Omron CX-Programmer project NewProject (CX-Programmer 9.75)

# PLC cj1m_cpu22: CJ1M CPU11

## Global symbols (name address type ; comment)
ActualPosition_Y _NCCPU204_ReadActualPosition_REAL
101.00 BOOL  ; Coolant Pump On
101.01 BOOL  ; X Lube Pump On
101.02 BOOL  ; Main Pump On
101.03 BOOL  ; Spindle Lube Pump On
101.04 BOOL  ; SP Main Contactor On
101.05 BOOL  ; SP Delta Contactor On
101.06 BOOL  ; SP Star Contactor On
101.07 BOOL  ; Work Light On
101.08 BOOL  ; Red Tower Light On
101.09 BOOL  ; Greeen Tower Light On
101.10 BOOL  ; Yellow Tower Light On
101.11 BOOL  ; X + Move Solenoid
101.12 BOOL  ; X - Move Solenoid
101.13 BOOL  ; X Slow Speed Solenoid
101.14 BOOL  ; X Pressure Relief Solenoid
102.00 BOOL  ; Table Magnet On
102.01 BOOL  ; Table Demagnet On
1.00 BOOL  ; Emergency PB
1.01 BOOL  ; X + PB
1.02 BOOL  ; X - PB
1.03 BOOL  ; X Stop PB
1.04 BOOL  ; Man/Auto SW
1.05 BOOL  ; Coolant Pump Overload Input
1.06 BOOL  ; X Lube Pump Overload Input
1.07 BOOL  ; Main Pump Overload Input
1.08 BOOL  ; Counterbalance Pump Overload Input
1.09 BOOL  ; Spindle Lube Pump Overload Input
1.10 BOOL  ; Spindle Chiller Overload Input
1.11 BOOL  ; Main Chiller Overload Input
1.14 BOOL  ; Alarm Y Axis Input
1.15 BOOL  ; Alarm Z Axis Input
2.00 BOOL  ; X Axis Handwheel Input
2.01 BOOL  ; Y Axis Handwheel Input
2.02 BOOL  ; Z Axis Handwheel Input
2.03 BOOL  ; X1 Speed Input
2.04 BOOL  ; X10 Speed Input
2.05 BOOL  ; X100 Speed Input
2.06 BOOL  ; X+ Work Limit SW
2.07 BOOL  ; X - Work Limit SW
2.08 BOOL  ; X + Safety Limit SW
2.09 BOOL  ; X - Safety Limit SW
2.10 BOOL  ; Z - Limit SW
2.11 BOOL  ; Z + Limit SW
2.12 BOOL  ; Z Zero Limit SW
2.13 BOOL  ; Y - Limit SW
2.14 BOOL  ; Y + Limit SW
2.15 BOOL  ; Y Zero Limit SW
3.00 BOOL  ; X Lube PR SW
3.01 BOOL  ; Spindle Lube PR SW
A540.08 BOOL  ; Y Axis Positive Limit
A540.09 BOOL  ; Y Axis Negative Limit
A541.08 BOOL  ; Z Axis Positive Limit
A541.09 BOOL  ; Z Axis Negative Limit
D10 CHANNEL  ; Travel Position
D100 CHANNEL  ; Axis Y Acceleration
D102 CHANNEL  ; Axis Y Deceleration
D108 CHANNEL  ; Axis Y Velocity
D110 CHANNEL  ; Y Actual Position
D112 CHANNEL  ; Y Jog Velocity
D20 CHANNEL  ; Travel Position Z Axis
D200 CHANNEL  ; Axis Z Acceleration
D202 CHANNEL  ; Axis Z Decceleration
D208 CHANNEL  ; Axis Z Velocity
D210 CHANNEL  ; Z Actual Position
D212 CHANNEL  ; Z Jog Velocity
W11.00 BOOL  ; Emergency Active
W11.01 BOOL  ; X + Move
W11.02 BOOL  ; X - Move
W11.03 BOOL  ; X Stop
W11.04 BOOL  ; Auto Mode
W11.05 BOOL  ; Coolant Pump Overload
W11.06 BOOL  ; X Lube Pump Overload
W11.07 BOOL  ; Main Pump Overload
W11.08 BOOL  ; Counterbalance Pump Overload
W11.09 BOOL  ; Spindle Lube Pump Overload
W11.10 BOOL  ; Spindle Chiller Overload
W11.11 BOOL  ; Main Chiller Overload
W11.14 BOOL  ; Alarm Y Axis
W11.15 BOOL  ; Alarm Z Axis
W12.00 BOOL  ; Handwheel X axis
W12.01 BOOL  ; Handwheel Y Axis
W12.02 BOOL  ; Handwheel Z Axis
W12.03 BOOL  ; Handwheel X1 Speed
W12.04 BOOL  ; Handwheel X10 Speed
W12.05 BOOL  ; Handwheel X100 Speed
W12.06 BOOL  ; X + Work Limit
W12.07 BOOL  ; X - Work Limit
W12.08 BOOL  ; X + Safety Limit
W12.09 BOOL  ; X - Safety Limit
W12.10 BOOL  ; Z - Limit
W12.11 BOOL  ; Z + Limit
W12.12 BOOL  ; Z Zero Limit
W12.13 BOOL  ; Y - Limit
W12.14 BOOL  ; Y + Limit
W12.15 BOOL  ; Y Zero Limit
W13.00 BOOL  ; X Lube Pressure Ok
W13.01 BOOL  ; Spindle Lube Pressure Ok
W21.00 BOOL  ; Coolant Pump On
W21.01 BOOL  ; X Lube Pump On
W21.02 BOOL  ; Main Pump On
W21.03 BOOL  ; Spindle Lube Pump On
W21.04 BOOL  ; Spindle Main Contactor On
W21.05 BOOL  ; Spindle Delta Contactor On
W21.06 BOOL  ; Spindle Star Contactor On
W21.07 BOOL  ; Work Light On
W21.08 BOOL  ; Red Tower Light
W21.09 BOOL  ; Green Tower Light
W21.10 BOOL  ; Yellow Tower Light
W21.11 BOOL  ; X + Move Command
W21.12 BOOL  ; X - Move Command
W21.13 BOOL  ; X Slow Speed Command
W21.14 BOOL  ; X Pressure Relief Command
W22.00 BOOL  ; Table Magnet On
W22.01 BOOL  ; Table Demagnet On
W30.00 BOOL  ; Y Axis Move Command
W30.04 BOOL  ; Y Axis Forward
W30.05 BOOL  ; Y Axis Backward
W31.04 BOOL  ; Z Jog Forward
W31.05 BOOL  ; Z Jog Backwards
W40.00 BOOL  ; X + Move Command
W40.01 BOOL  ; X - Move Command
W40.02 BOOL  ; X + Move Manual
W40.03 BOOL  ; X - Move Manual
JogBackwards_Y _NCCPU030_MoveVelocity_REAL
JogBackwards_Z _NCCPU030_MoveVelocity_REAL
JogForward_Y _NCCPU030_MoveVelocity_REAL
JogForward_Z _NCCPU030_MoveVelocity_REAL
MoveAbsolute_Z _NCCPU010_MoveAbsolute_REAL
MoveY _NCCPU010_MoveAbsolute_REAL
Position_Z _NCCPU204_ReadActualPosition_REAL

## Program NewProgram1 (cyclic task 0)

### Section Inputs

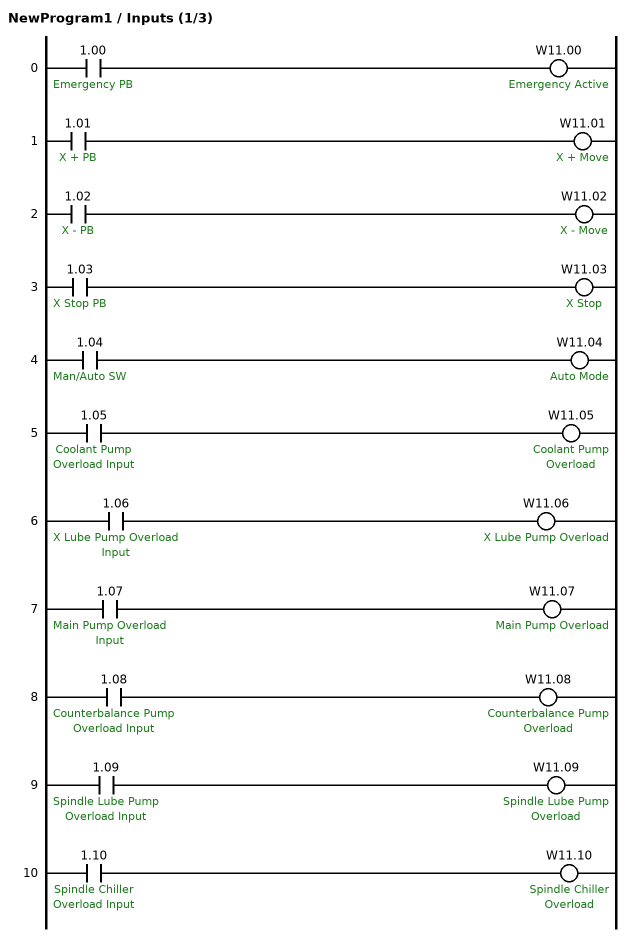
; rung 0
LD 1.00  ; Emergency PB
OUT W11.00  ; Emergency Active
; rung 1
LD 1.01  ; X + PB
OUT W11.01  ; X + Move
; rung 2
LD 1.02  ; X - PB
OUT W11.02  ; X - Move
; rung 3
LD 1.03  ; X Stop PB
OUT W11.03  ; X Stop
; rung 4
LD 1.04  ; Man/Auto SW
OUT W11.04  ; Auto Mode
; rung 5
LD 1.05  ; Coolant Pump Overload Input
OUT W11.05  ; Coolant Pump Overload
; rung 6
LD 1.06  ; X Lube Pump Overload Input
OUT W11.06  ; X Lube Pump Overload
; rung 7
LD 1.07  ; Main Pump Overload Input
OUT W11.07  ; Main Pump Overload
; rung 8
LD 1.08  ; Counterbalance Pump Overload Input
OUT W11.08  ; Counterbalance Pump Overload
; rung 9
LD 1.09  ; Spindle Lube Pump Overload Input
OUT W11.09  ; Spindle Lube Pump Overload
; rung 10
LD 1.10  ; Spindle Chiller Overload Input
OUT W11.10  ; Spindle Chiller Overload

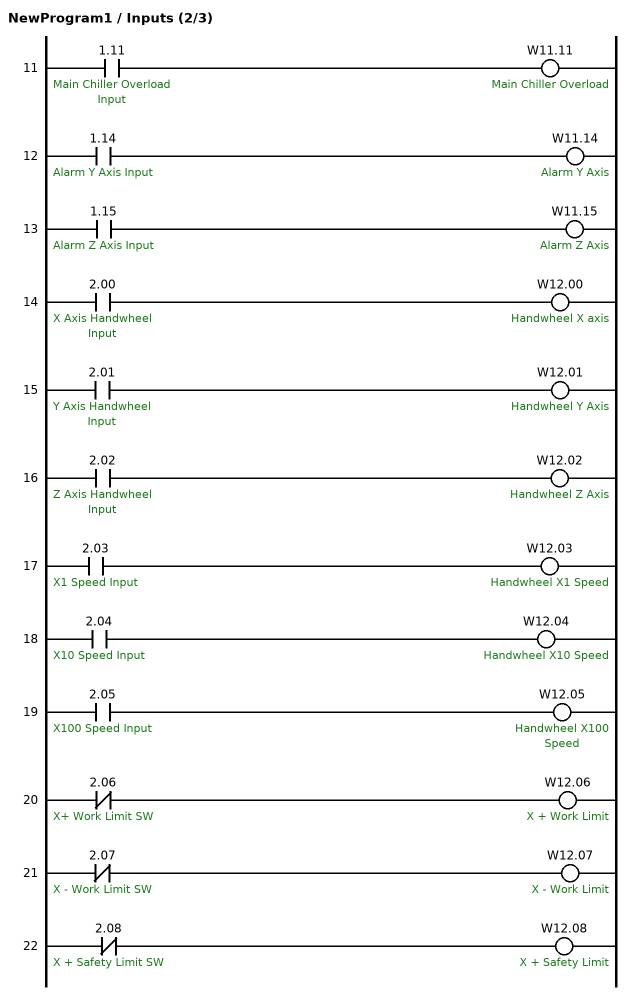
; rung 11
LD 1.11  ; Main Chiller Overload Input
OUT W11.11  ; Main Chiller Overload
; rung 12
LD 1.14  ; Alarm Y Axis Input
OUT W11.14  ; Alarm Y Axis
; rung 13
LD 1.15  ; Alarm Z Axis Input
OUT W11.15  ; Alarm Z Axis
; rung 14
LD 2.00  ; X Axis Handwheel Input
OUT W12.00  ; Handwheel X axis
; rung 15
LD 2.01  ; Y Axis Handwheel Input
OUT W12.01  ; Handwheel Y Axis
; rung 16
LD 2.02  ; Z Axis Handwheel Input
OUT W12.02  ; Handwheel Z Axis
; rung 17
LD 2.03  ; X1 Speed Input
OUT W12.03  ; Handwheel X1 Speed
; rung 18
LD 2.04  ; X10 Speed Input
OUT W12.04  ; Handwheel X10 Speed
; rung 19
LD 2.05  ; X100 Speed Input
OUT W12.05  ; Handwheel X100 Speed
; rung 20
LDNOT 2.06  ; X+ Work Limit SW
OUT W12.06  ; X + Work Limit
; rung 21
LDNOT 2.07  ; X - Work Limit SW
OUT W12.07  ; X - Work Limit
; rung 22
LDNOT 2.08  ; X + Safety Limit SW
OUT W12.08  ; X + Safety Limit

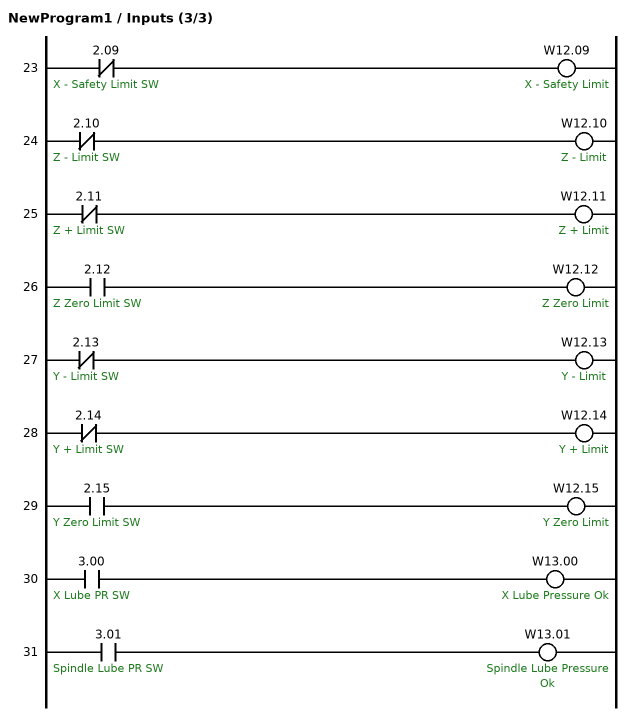
; rung 23
LDNOT 2.09  ; X - Safety Limit SW
OUT W12.09  ; X - Safety Limit
; rung 24
LDNOT 2.10  ; Z - Limit SW
OUT W12.10  ; Z - Limit
; rung 25
LDNOT 2.11  ; Z + Limit SW
OUT W12.11  ; Z + Limit
; rung 26
LD 2.12  ; Z Zero Limit SW
OUT W12.12  ; Z Zero Limit
; rung 27
LDNOT 2.13  ; Y - Limit SW
OUT W12.13  ; Y - Limit
; rung 28
LDNOT 2.14  ; Y + Limit SW
OUT W12.14  ; Y + Limit
; rung 29
LD 2.15  ; Y Zero Limit SW
OUT W12.15  ; Y Zero Limit
; rung 30
LD 3.00  ; X Lube PR SW
OUT W13.00  ; X Lube Pressure Ok
; rung 31
LD 3.01  ; Spindle Lube PR SW
OUT W13.01  ; Spindle Lube Pressure Ok

### Section Outputs

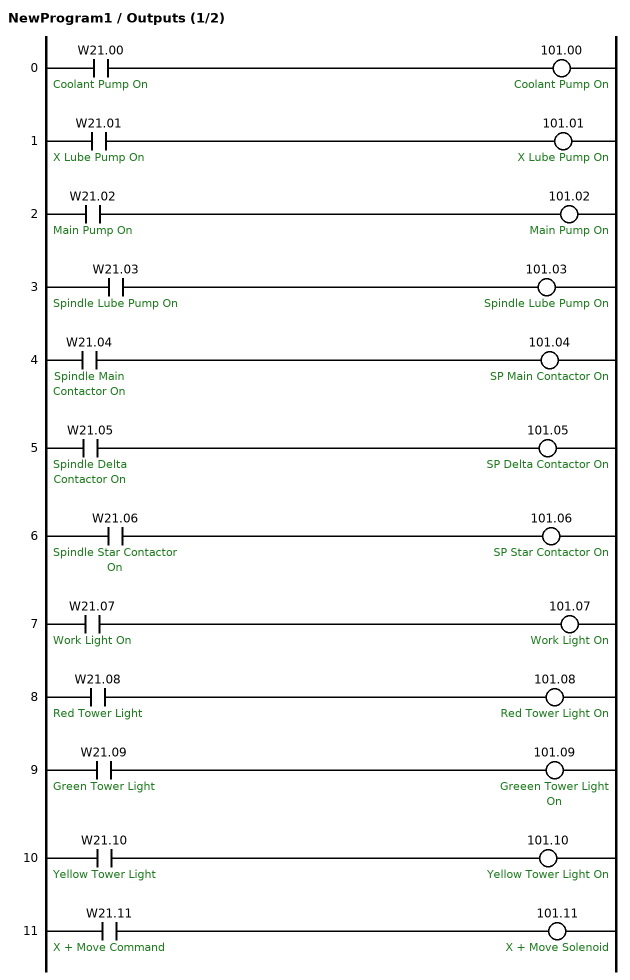
; rung 0
LD W21.00  ; Coolant Pump On
OUT 101.00  ; Coolant Pump On
; rung 1
LD W21.01  ; X Lube Pump On
OUT 101.01  ; X Lube Pump On
; rung 2
LD W21.02  ; Main Pump On
OUT 101.02  ; Main Pump On
; rung 3
LD W21.03  ; Spindle Lube Pump On
OUT 101.03  ; Spindle Lube Pump On
; rung 4
LD W21.04  ; Spindle Main Contactor On
OUT 101.04  ; SP Main Contactor On
; rung 5
LD W21.05  ; Spindle Delta Contactor On
OUT 101.05  ; SP Delta Contactor On
; rung 6
LD W21.06  ; Spindle Star Contactor On
OUT 101.06  ; SP Star Contactor On
; rung 7
LD W21.07  ; Work Light On
OUT 101.07  ; Work Light On
; rung 8
LD W21.08  ; Red Tower Light
OUT 101.08  ; Red Tower Light On
; rung 9
LD W21.09  ; Green Tower Light
OUT 101.09  ; Greeen Tower Light On
; rung 10
LD W21.10  ; Yellow Tower Light
OUT 101.10  ; Yellow Tower Light On
; rung 11
LD W21.11  ; X + Move Command
OUT 101.11  ; X + Move Solenoid

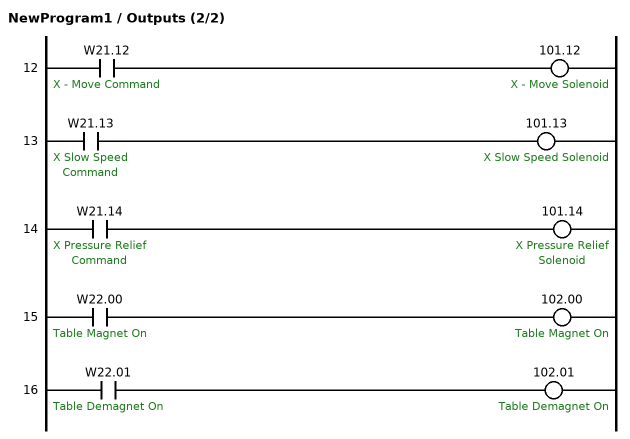
; rung 12
LD W21.12  ; X - Move Command
OUT 101.12  ; X - Move Solenoid
; rung 13
LD W21.13  ; X Slow Speed Command
OUT 101.13  ; X Slow Speed Solenoid
; rung 14
LD W21.14  ; X Pressure Relief Command
OUT 101.14  ; X Pressure Relief Solenoid
; rung 15
LD W22.00  ; Table Magnet On
OUT 102.00  ; Table Magnet On
; rung 16
LD W22.01  ; Table Demagnet On
OUT 102.01  ; Table Demagnet On

### Section Table_Movement

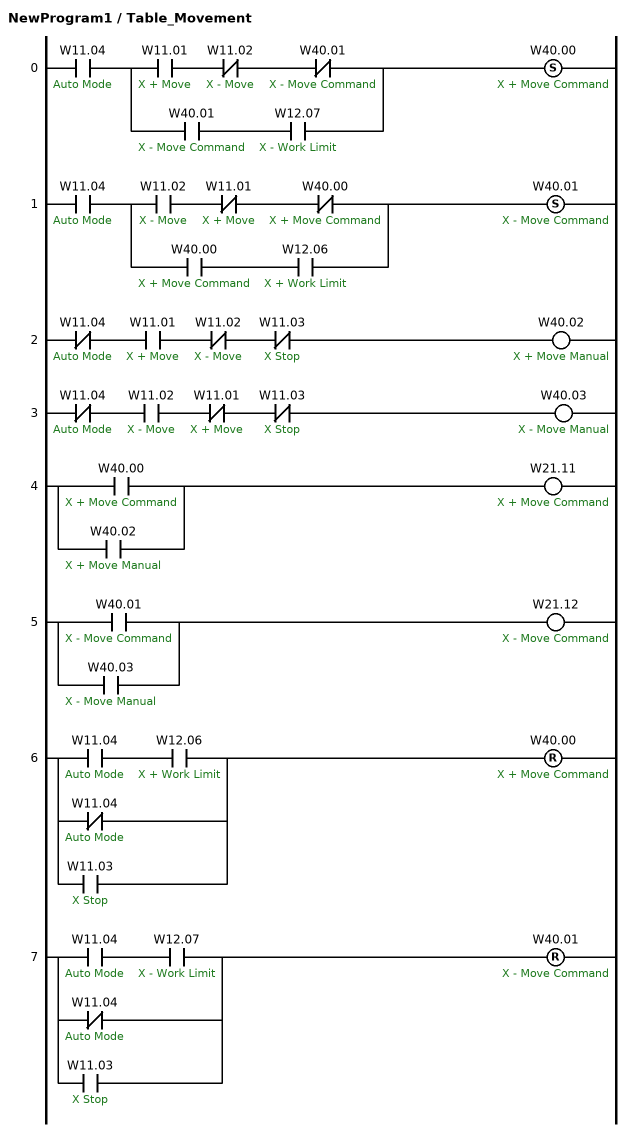
; rung 0
LD W11.04  ; Auto Mode
LD W11.01  ; X + Move
ANDNOT W11.02  ; X - Move
ANDNOT W40.01  ; X - Move Command
LD W40.01  ; X - Move Command
AND W12.07  ; X - Work Limit
ORLD
ANDLD
SET W40.00  ; X + Move Command
; rung 1
LD W11.04  ; Auto Mode
LD W11.02  ; X - Move
ANDNOT W11.01  ; X + Move
ANDNOT W40.00  ; X + Move Command
LD W40.00  ; X + Move Command
AND W12.06  ; X + Work Limit
ORLD
ANDLD
SET W40.01  ; X - Move Command
; rung 2
LDNOT W11.04  ; Auto Mode
AND W11.01  ; X + Move
ANDNOT W11.02  ; X - Move
ANDNOT W11.03  ; X Stop
OUT W40.02  ; X + Move Manual
; rung 3
LDNOT W11.04  ; Auto Mode
AND W11.02  ; X - Move
ANDNOT W11.01  ; X + Move
ANDNOT W11.03  ; X Stop
OUT W40.03  ; X - Move Manual
; rung 4
LD W40.00  ; X + Move Command
OR W40.02  ; X + Move Manual
OUT W21.11  ; X + Move Command
; rung 5
LD W40.01  ; X - Move Command
OR W40.03  ; X - Move Manual
OUT W21.12  ; X - Move Command
; rung 6
LD W11.04  ; Auto Mode
AND W12.06  ; X + Work Limit
ORNOT W11.04  ; Auto Mode
OR W11.03  ; X Stop
RSET W40.00  ; X + Move Command
; rung 7
LD W11.04  ; Auto Mode
AND W12.07  ; X - Work Limit
ORNOT W11.04  ; Auto Mode
OR W11.03  ; X Stop
RSET W40.01  ; X - Move Command

### Section Axis_Y

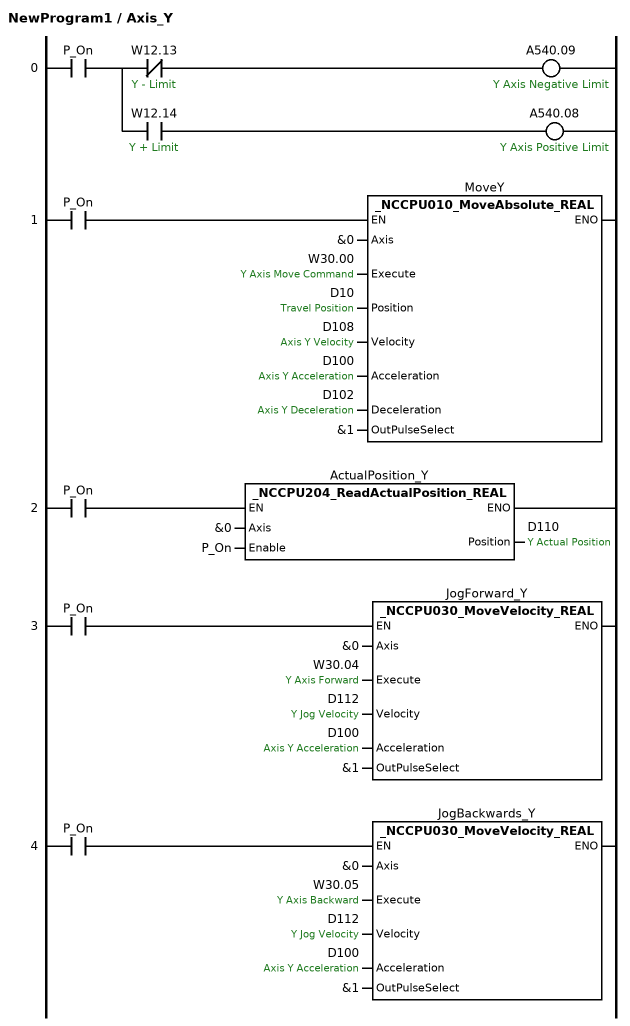
; rung 0
LD P_On
OUT TR0
ANDNOT W12.13  ; Y - Limit
OUT A540.09  ; Y Axis Negative Limit
LD TR0
AND W12.14  ; Y + Limit
OUT A540.08  ; Y Axis Positive Limit
; rung 1
LD P_On
CALL MoveY : _NCCPU010_MoveAbsolute_REAL (Axis := &0, Execute := W30.00, Position := D10, Velocity := D108, Acceleration := D100, Deceleration := D102, OutPulseSelect := &1)  ; Y Axis Move Command, Travel Position, Axis Y Velocity, Axis Y Acceleration, Axis Y Deceleration
; rung 2
LD P_On
CALL ActualPosition_Y : _NCCPU204_ReadActualPosition_REAL (Axis := &0, Enable := P_On, Position => D110)  ; Y Actual Position
; rung 3
LD P_On
CALL JogForward_Y : _NCCPU030_MoveVelocity_REAL (Axis := &0, Execute := W30.04, Velocity := D112, Acceleration := D100, OutPulseSelect := &1)  ; Y Axis Forward, Y Jog Velocity, Axis Y Acceleration
; rung 4
LD P_On
CALL JogBackwards_Y : _NCCPU030_MoveVelocity_REAL (Axis := &0, Execute := W30.05, Velocity := D112, Acceleration := D100, OutPulseSelect := &1)  ; Y Axis Backward, Y Jog Velocity, Axis Y Acceleration

### Section Axis_Z

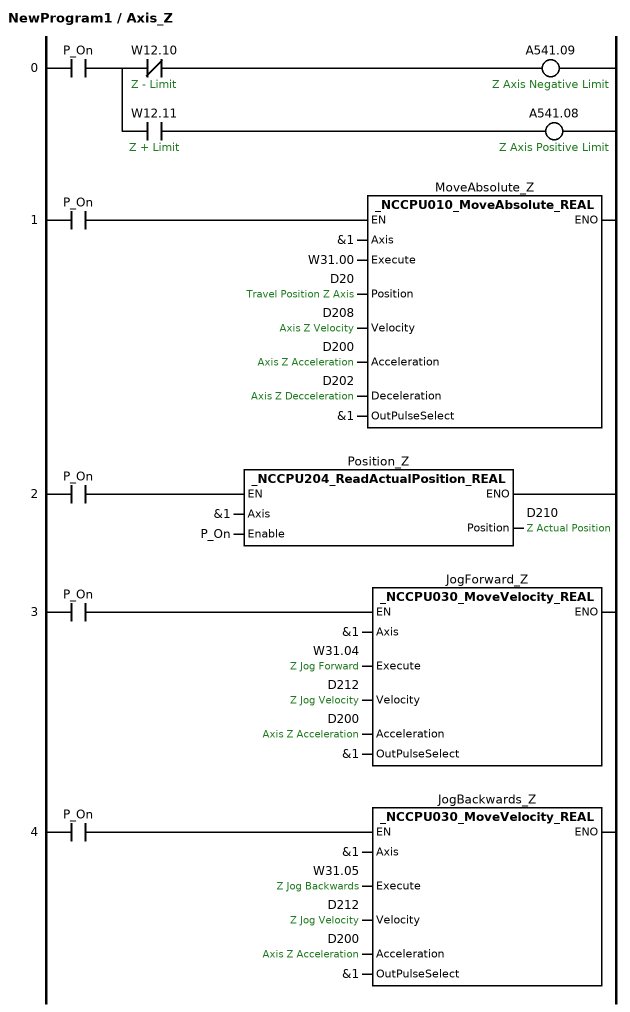
; rung 0
LD P_On
OUT TR0
ANDNOT W12.10  ; Z - Limit
OUT A541.09  ; Z Axis Negative Limit
LD TR0
AND W12.11  ; Z + Limit
OUT A541.08  ; Z Axis Positive Limit
; rung 1
LD P_On
CALL MoveAbsolute_Z : _NCCPU010_MoveAbsolute_REAL (Axis := &1, Execute := W31.00, Position := D20, Velocity := D208, Acceleration := D200, Deceleration := D202, OutPulseSelect := &1)  ; Travel Position Z Axis, Axis Z Velocity, Axis Z Acceleration, Axis Z Decceleration
; rung 2
LD P_On
CALL Position_Z : _NCCPU204_ReadActualPosition_REAL (Axis := &1, Enable := P_On, Position => D210)  ; Z Actual Position
; rung 3
LD P_On
CALL JogForward_Z : _NCCPU030_MoveVelocity_REAL (Axis := &1, Execute := W31.04, Velocity := D212, Acceleration := D200, OutPulseSelect := &1)  ; Z Jog Forward, Z Jog Velocity, Axis Z Acceleration
; rung 4
LD P_On
CALL JogBackwards_Z : _NCCPU030_MoveVelocity_REAL (Axis := &1, Execute := W31.05, Velocity := D212, Acceleration := D200, OutPulseSelect := &1)  ; Z Jog Backwards, Z Jog Velocity, Axis Z Acceleration

### Section END
; rung 0
END(001)

## Function block _NCCPU010_MoveAbsolute_REAL (Omron library block, body left out)

## Function block _NCCPU030_MoveVelocity_REAL (Omron library block, body left out)

## Function block _NCCPU204_ReadActualPosition_REAL (Omron library block, body left out)